// TIA Portal project "chain_transportation_conveyor_V17" (V17)

(* hardware
DEVICE "S7-1200 station_1"  S7-1200 Station
   slot 0: "Rack_0"  S7-1200 Rack  Rack  V1.0
   slot 1: "PLC_1"  CPU 1215C DC/DC/DC  6ES7 215-1AG40-0XB0  V4.2
DEVICE "Touchpanel"  TP700 Comfort
   slot 0: "Touchpanel"  TP700 Comfort  6AV2 124-0GC01-0AX0  15.0.0.0
   slot 1: "HMI_RT_1"  TP700 Comfort  6AV2 124-0GC01-0AX0  15.0.0.0
   slot 5: "Touchpanel.IE_CP_1"  PROFINET Interface  15.0.0.0
      slot 1: "PROFINET Interface_1"  PROFINET Interface
         slot 1: "Port_1"  Port
         slot 2: "Port_2"  Port
   slot 7: "Touchpanel.MPI/DP_CP_1"  MPI/DP Interface  15.0.0.0
*)

// ===== PLC "PLC_1"  CPU 1215C DC/DC/DC =====

VAR_GLOBAL   // PLC tag table "Default tag table"
   "stop" AT %M0.1 : Bool;
   "start" AT %M0.0 : Bool;
   "start_mem" AT %M0.2 : Bool;
   "sensor_1" AT %M0.3 : Bool;
   "sensor_2" AT %M0.4 : Bool;
   "conveyor_1" AT %Q0.0 : Bool;
   "chain_height" AT %Q0.1 : Bool;
   "sensor_3" AT %M0.5 : Bool;
   "conveyor_2" AT %Q0.2 : Bool;
   "conveyor_3" AT %Q0.3 : Bool;
   "chain_motor(1)" AT %Q0.4 : Bool;
   "chain_sensor_1" AT %M0.6 : Bool;
   "chain_sensor_2" AT %M0.7 : Bool;
END_VAR

DATA_BLOCK "chain_conveyor_DB"   // DB1
{ S7_Optimized_Access := 'TRUE' }
VERSION : 0.1
// stored: InstanceOfName chain_conveyor
"chain_conveyor"
BEGIN
END_DATA_BLOCK

DATA_BLOCK "chain_conveyor_DB_1"   // DB2
{ S7_Optimized_Access := 'TRUE' }
VERSION : 0.1
// stored: InstanceOfName chain_conveyor
"chain_conveyor"
BEGIN
END_DATA_BLOCK

DATA_BLOCK "chain_conveyor_DB_2"   // DB3
{ S7_Optimized_Access := 'TRUE' }
VERSION : 0.1
// stored: InstanceOfName chain_conveyor
"chain_conveyor"
BEGIN
END_DATA_BLOCK

DATA_BLOCK "chain_motor_DB"   // DB4
{ S7_Optimized_Access := 'TRUE' }
VERSION : 0.1
// stored: InstanceOfName chain_motor
"chain_motor"
BEGIN
END_DATA_BLOCK

FUNCTION_BLOCK "chain_conveyor"   // FB1, LAD
{ S7_Optimized_Access := 'TRUE' }
VERSION : 0.1
   VAR_INPUT
      prev_sensor : Bool;
      curr_sensor : Bool;
      next_sensor : Bool;
      chain_sensor_1 : Bool;
      chain_sensor_2 : Bool;
   END_VAR
   VAR_OUTPUT
      conveyor : Bool;
      chain_height : Bool;
      chain_motor : Bool;
   END_VAR
   VAR
      run_motor_2 : Bool;
      run_motor : Bool;
      IEC_Timer_0_Instance : TON_TIME;
      IEC_Timer_0_Instance_1 : TOF_TIME;
      IEC_Timer_0_Instance_2 : TOF_TIME;
   END_VAR
BEGIN

REGION Network 1
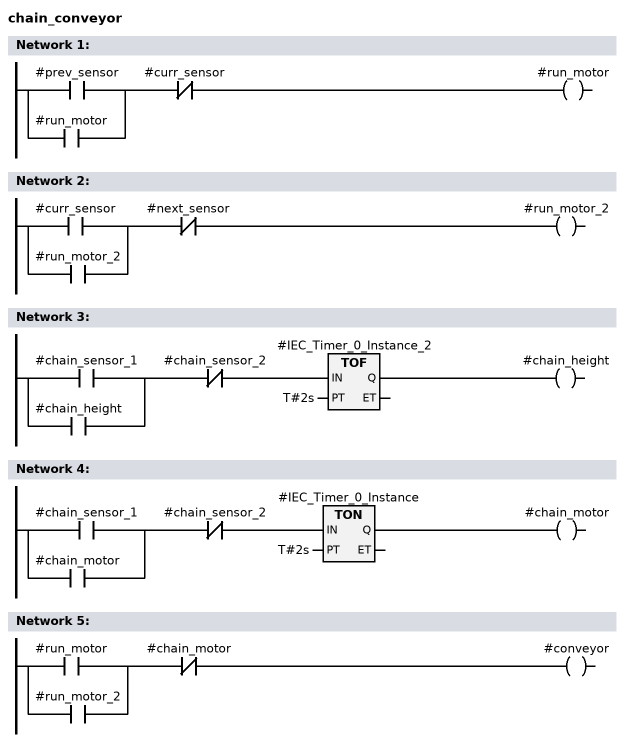
   RUNG wire#powerrail
      Contact( #prev_sensor )
      wire#w1
      I_Contact( #curr_sensor )
      Coil( #run_motor )
   END_RUNG
   RUNG wire#powerrail
      Contact( #run_motor )
   END_RUNG wire#w1
   // the same network as SCL:
   #run_motor := (#prev_sensor OR #run_motor) AND NOT #curr_sensor;
END_REGION

REGION Network 2
   RUNG wire#powerrail
      Contact( #curr_sensor )
      wire#w1
      I_Contact( #next_sensor )
      Coil( #run_motor_2 )
   END_RUNG
   RUNG wire#powerrail
      Contact( #run_motor_2 )
   END_RUNG wire#w1
   // the same network as SCL:
   #run_motor_2 := (#curr_sensor OR #run_motor_2) AND NOT #next_sensor;
END_REGION

REGION Network 3
   #IEC_Timer_0_Instance_2(IN := (#chain_sensor_1 OR #chain_height) AND NOT #chain_sensor_2, PT := T#2s);   // TOF
   #chain_height := #IEC_Timer_0_Instance_2.Q;
END_REGION

REGION Network 4
   #IEC_Timer_0_Instance(IN := (#chain_sensor_1 OR #chain_motor) AND NOT #chain_sensor_2, PT := T#2s);   // TON
   #chain_motor := #IEC_Timer_0_Instance.Q;
END_REGION

REGION Network 5
   RUNG wire#powerrail
      Contact( #run_motor )
      wire#w1
      I_Contact( #chain_motor )
      Coil( #conveyor )
   END_RUNG
   RUNG wire#powerrail
      Contact( #run_motor_2 )
   END_RUNG wire#w1
   // the same network as SCL:
   #conveyor := (#run_motor OR #run_motor_2) AND NOT #chain_motor;
END_REGION
END_FUNCTION_BLOCK

FUNCTION_BLOCK "chain_motor"   // FB2, LAD
{ S7_Optimized_Access := 'TRUE' }
VERSION : 0.1
   VAR_INPUT
      curr_sensor : Bool;
      next_sensor : Bool;
   END_VAR
   VAR_OUTPUT
      chain_height : Bool;
      chain_motor : Bool;
   END_VAR
BEGIN

REGION Network 1
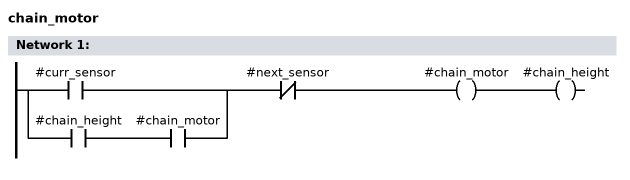
   RUNG wire#powerrail
      Contact( #curr_sensor )
      wire#w1
      I_Contact( #next_sensor )
      Coil( #chain_motor )
      Coil( #chain_height )
   END_RUNG
   RUNG wire#powerrail
      Contact( #chain_height )
      Contact( #chain_motor )
   END_RUNG wire#w1
   // the same network as SCL:
   #chain_motor := (#curr_sensor OR (#chain_height AND #chain_motor)) AND NOT #next_sensor;
   #chain_height := #chain_motor;
END_REGION
END_FUNCTION_BLOCK

ORGANIZATION_BLOCK "Main"   // OB1, LAD, ProgramCycle
TITLE = "Main Program Sweep (Cycle)"
{ S7_Optimized_Access := 'TRUE' }
VERSION : 0.1
   VAR_INPUT
      Initial_Call : Bool;   // Initial call of this OB
      Remanence : Bool;   // =True, if remanent data are available
   END_VAR
   VAR_TEMP   // added for the SCL form of the ladder/FBD networks
      _w1 : Bool;
   END_VAR
BEGIN

REGION Network 1
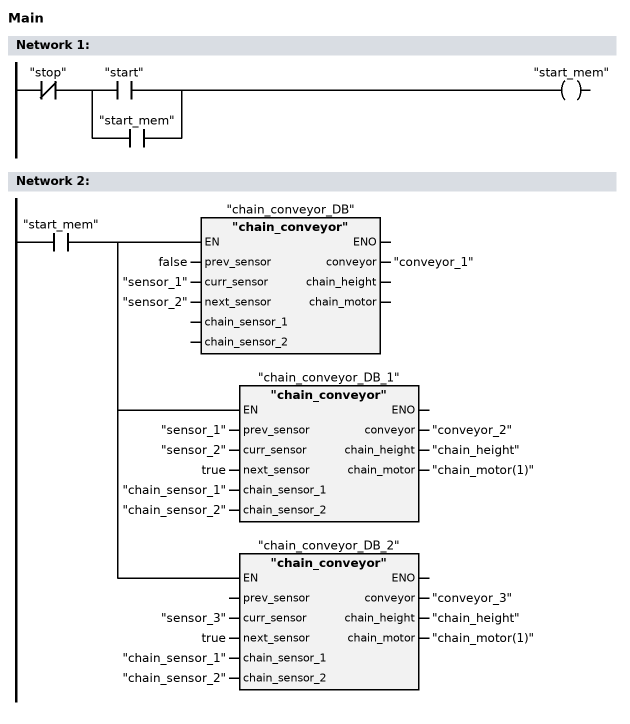
   RUNG wire#powerrail
      I_Contact( "stop" )
      wire#w1
      Contact( "start" )
      wire#w2
      Coil( "start_mem" )
   END_RUNG
   RUNG wire#w1
      Contact( "start_mem" )
   END_RUNG wire#w2
   // the same network as SCL:
   "start_mem" := NOT "stop" AND ("start" OR "start_mem");
END_REGION

REGION Network 2
   RUNG wire#powerrail
      Contact( "start_mem" )
      wire#w1
      "chain_conveyor_DB"(prev_sensor := false, curr_sensor := "sensor_1", next_sensor := "sensor_2", chain_sensor_1 :=, chain_sensor_2 :=, conveyor => "conveyor_1", chain_height =>, chain_motor =>)
   END_RUNG
   RUNG wire#w1
      "chain_conveyor_DB_1"(prev_sensor := "sensor_1", curr_sensor := "sensor_2", next_sensor := true, chain_sensor_1 := "chain_sensor_1", chain_sensor_2 := "chain_sensor_2", conveyor => "conveyor_2", chain_height => "chain_height", chain_motor => "chain_motor(1)")
   END_RUNG
   RUNG wire#w1
      "chain_conveyor_DB_2"(prev_sensor :=, curr_sensor := "sensor_3", next_sensor := true, chain_sensor_1 := "chain_sensor_1", chain_sensor_2 := "chain_sensor_2", conveyor => "conveyor_3", chain_height => "chain_height", chain_motor => "chain_motor(1)")
   END_RUNG
   // the same network as SCL:
   #_w1 := "start_mem";
   IF #_w1 THEN
       "chain_conveyor_DB"(prev_sensor := false,   // "chain_conveyor"
                           curr_sensor := "sensor_1",
                           next_sensor := "sensor_2",
                           conveyor => "conveyor_1");
       "chain_conveyor_DB_1"(prev_sensor := "sensor_1",   // "chain_conveyor"
                             curr_sensor := "sensor_2",
                             next_sensor := true,
                             chain_sensor_1 := "chain_sensor_1",
                             chain_sensor_2 := "chain_sensor_2",
                             conveyor => "conveyor_2",
                             chain_height => "chain_height",
                             chain_motor => "chain_motor(1)");
       "chain_conveyor_DB_2"(curr_sensor := "sensor_3",   // "chain_conveyor"
                             next_sensor := true,
                             chain_sensor_1 := "chain_sensor_1",
                             chain_sensor_2 := "chain_sensor_2",
                             conveyor => "conveyor_3",
                             chain_height => "chain_height",
                             chain_motor => "chain_motor(1)");
   END_IF;
END_REGION
END_ORGANIZATION_BLOCK

(* ===== HMI "HMI_RT_1" =====
connection "HMI_Connection_1": ETHERNET, S7_1200_OMS

screen "Screen_1" 800x480
   Button "Button_1" at 11,440 size 96x32; TextOff 'Start'
   Button "Button_2" at 119,440 size 96x32; TextOff 'Stop'
   TextField "Text field_1" at 304,82 size 106x23; Text 'Conveyor 1'
   TextField "Text field_2" at 303,142 size 106x23; Text 'Conveyor 2'
   TextField "Text field_3" at 302,196 size 106x23; Text 'Conveyor 3'
   TextField "Text field_4" at 540,82 size 122x23; Text 'Chain Height'
   TextField "Text field_5" at 540,141 size 115x23; Text 'Chain Motor'
   TextField "Text field_6" at 75,83 size 83x23; Text 'Sensor 1'
   TextField "Text field_7" at 74,143 size 83x23; Text 'Sensor 2'
   TextField "Text field_8" at 73,197 size 83x23; Text 'Sensor 3'
*)